FUNCTION_BLOCK CounterTimer
VAR_INPUT
	fValue : REAL;
END_VAR
VAR
	values: ARRAY[0 .. globals.MAX_BUFFER_LENGTH] OF REAL;
	fValueSum: REAL := 0;
	fValueAverage: REAL := 0;
	
	nScanTotal: UDINT := 1;
	nLatencyCycles: UDINT := 0;
	nAccumCycles: UDINT := 100;
	
	nScanIndex: UDINT := 0;
	nWaitIndex: UDINT := 0;
	nAccumIndex: UDINT := 0;
	
	eState: CounterState:=CounterState.STOP;
	nState: INT; // for pyads, since it can't read the enum value properly
END_VAR

// Value counter and buffer. Performs consecutive measurements with
// configurable integration time and delay between measurements.

ProcessValue(fValue);
nState := eState;

METHOD PrepareMeasurement
VAR_INPUT
	nAccumMilliseconds: UDINT;
	nDelayMilliseconds: UDINT;
	nMeasurements: UDINT;
END_VAR
VAR
	nCyclesPerMillisecond: UDINT;
END_VAR
// CycleTime is in multiples of 100 ns
nCyclesPerMillisecond := 10_000 / getTaskCycleTime();

nScanTotal := LIMIT(1, nMeasurements, globals.MAX_BUFFER_LENGTH);
nAccumCycles := MAX(1, nAccumMilliseconds * nCyclesPerMillisecond);
nLatencyCycles := nDelayMilliseconds * nCyclesPerMillisecond;
END_METHOD

METHOD ProcessValue
VAR_INPUT
	fValue : REAL;
END_VAR
// integrate values for given number of ticks, then store average
// enter wait loop after storing

IF eState = CounterState.MEASURE THEN
	fValueSum := fValueSum + fValue;
	nAccumIndex := nAccumIndex + 1;
	fValueAverage := fValueSum / UDINT_TO_REAL(nAccumIndex);

	IF nAccumIndex >= nAccumCycles THEN
		values[nScanIndex] := fValueAverage;
		nScanIndex := nScanIndex + 1;
		nAccumIndex := 0;
		fValueSum := 0;
		
		IF nScanIndex >= nScanTotal THEN
			eState := CounterState.STOP;
		ELSE
			eState := CounterState.WAIT;
			nWaitIndex := 0;	
		END_IF
	END_IF
END_IF

IF eState = CounterState.WAIT THEN
	IF nWaitIndex >= nLatencyCycles THEN
		eState := CounterState.MEASURE;			
	ELSE
		nWaitIndex := nWaitIndex + 1;
	END_IF
END_IF
END_METHOD

METHOD StartBuffer
eState := CounterState.MEASURE;
nScanIndex := 0;
nWaitIndex := 0;
nAccumIndex := 0;
fValueSum := 0;
END_METHOD

METHOD StopBuffer
eState := CounterState.STOP;
END_METHOD

END_FUNCTION_BLOCK

(* stored: Version 1.1.0.1, ProductVersion 3.1.4024.15
   POU CounterTimer: Id {538a4290-1fe2-4f16-8415-445ed81e1156}, SpecialFunc None
   Method PrepareMeasurement: Id {b0ddb6e3-5a83-4b0b-aa50-e0a4e6428f6d}
   Method ProcessValue: Id {fcef7e0b-4b79-4ad0-9a17-31eb21a8b8aa}
   Method StartBuffer: Id {6adea8aa-27b8-4149-8c81-b4583f5d2607}
   Method StopBuffer: Id {3921f370-7734-4c53-aee6-52fa9ffae7f6} *)
